Yaskawa INFORM job: s2D_Face_left.JBI

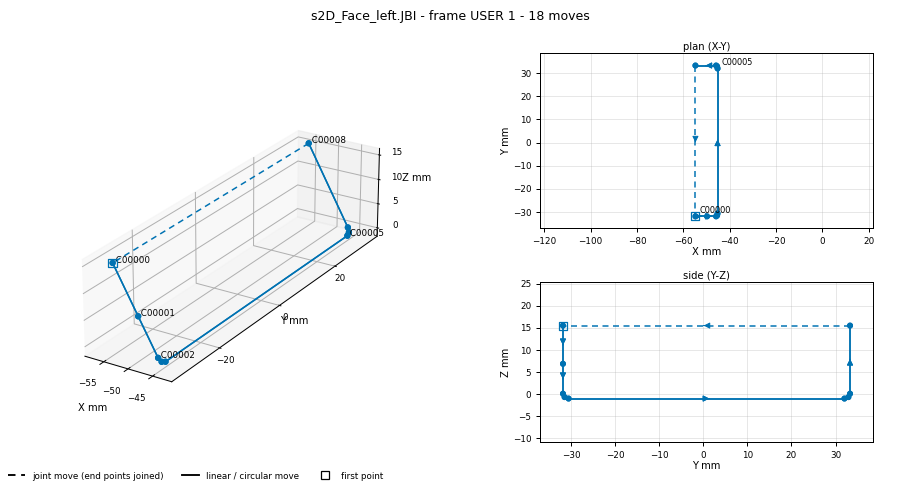
[picture p0: tool path of s2D_Face_left.JBI in frame USER 1, 18 of 18 moves have a stored position in this frame; points joined in program order, loops and branches not executed]
/JOB
//NAME s2D_Face_left
//POS
///NPOS 9,0,0,0,0,0
///USER 1
///TOOL 8
///POSTYPE USER
///RECTAN
///RCONF 1,0,0,0,0,0
C00000=53.984,-29.817,15.539,-90.000,-150.794,-116.565
C00001=53.984,-24.817,6.879,-90.000,-150.794,-116.565
C00002=53.984,-20.744,-0.175,-90.000,-150.794,-116.565
C00003=53.705,-20.407,-0.758,-90.000,-150.794,-116.565
C00004=53.031,-20.268,-1.000,-90.000,-150.794,-116.565
C00005=-55.536,-20.268,-1.000,-90.000,-150.794,-116.565
C00006=-56.209,-20.407,-0.758,-90.000,-150.794,-116.565
C00007=-56.488,-20.744,-0.175,-90.000,-150.794,-116.565
C00008=-56.488,-29.817,15.539,-90.000,-150.794,-116.565
C00000=-54.817,-31.806,15.539,180.000,-152.507,146.310
C00001=-49.817,-31.806,6.879,180.000,-152.507,146.310
C00002=-45.903,-31.806,0.100,180.000,-152.507,146.310
C00003=-45.454,-31.434,-0.678,180.000,-152.507,146.310
C00004=-45.268,-30.536,-1.000,180.000,-152.507,146.310
C00005=-45.268,32.000,-1.000,180.000,-152.507,146.310
C00006=-45.454,32.898,-0.678,180.000,-152.507,146.310
C00007=-45.903,33.270,0.100,180.000,-152.507,146.310
C00008=-54.817,33.270,15.539,180.000,-152.507,146.310
//INST
///ATTR SC,RW,RJ
////FRAME USER 1
///GROUP1 RB1
///LVARS 2,0,0,0,0,0,0,0
NOP
SET LB000 1
SET LB001 25
MOVJ C00000 VJ=17
MOVL C00001 V=17 PL=LB000 ACC=LB001 DEC=LB001
' Plunge Move Starts
MOVL C00002 V=8 PL=LB000 ACC=LB001 DEC=LB001
' Lead In Move Starts
MOVL C00003 V=17 PL=LB000 ACC=LB001 DEC=LB001
MOVL C00004 V=17 PL=LB000 ACC=LB001 DEC=LB001
' Cutting Move Starts
MOVL C00005 V=17 PL=LB000 ACC=LB001 DEC=LB001
' Lead Out Move Starts
MOVL C00006 V=17 PL=LB000 ACC=LB001 DEC=LB001
MOVL C00007 V=17 PL=LB000 ACC=LB001 DEC=LB001
' Rapid Move Starts
MOVL C00008 V=17 PL=LB000 ACC=LB001 DEC=LB001
' By Autodesk Fusion CAM 2.0.20494
' Tool = 2
' Spindle = 5000 RPM
' Set Position Level
' Set Acceleration
' Program Start
' First Toolpath Point
' Last Toolpath Point
MOVJ C00000 VJ=17
MOVL C00001 V=17 PL=LB000 ACC=LB001 DEC=LB001
' Plunge Move Starts
MOVL C00002 V=8 PL=LB000 ACC=LB001 DEC=LB001
' Lead In Move Starts
MOVL C00003 V=17 PL=LB000 ACC=LB001 DEC=LB001
MOVL C00004 V=17 PL=LB000 ACC=LB001 DEC=LB001
' Cutting Move Starts
MOVL C00005 V=17 PL=LB000 ACC=LB001 DEC=LB001
' Lead Out Move Starts
MOVL C00006 V=17 PL=LB000 ACC=LB001 DEC=LB001
MOVL C00007 V=17 PL=LB000 ACC=LB001 DEC=LB001
' Rapid Move Starts
MOVL C00008 V=17 PL=LB000 ACC=LB001 DEC=LB001
' By Autodesk Fusion CAM 2.0.20494
' Tool = 8
' Spindle = 6000 RPM
' Set Position Level
' Set Acceleration
' Program Start
' First Toolpath Point
END
